TYPE S_ILValues_To_PC_Struct :
STRUCT
	PARAM000:REAL ;// 注入线法拉第筒温度节点01（℃） 
	PARAM001:REAL ;// 内靶温度节点02（℃） 
	PARAM002:REAL ;// 引出法拉第筒温度节点03（℃） 
	PARAM003:REAL ;// 温度节点04（℃） 
	PARAM004:REAL ;// 温度节点05（℃）
	PARAM005:REAL ;// 温度节点06（℃） 
	PARAM006:REAL ;// 温度节点07（℃） 
	PARAM007:REAL ;// 温度节点08（℃） 
	PARAM008:BOOL ;// 已经移去接地 
	PARAM009:BOOL ;// 地坑栅栏门已经关闭 
	PARAM010:BOOL ;// 加速器已合盖 
	PARAM011:BOOL ;// 无源节点01 
	PARAM012:BOOL ;// 无源节点02 
	PARAM013:BOOL ;// 离子源角阀2联锁开 
	PARAM014:BOOL ;// 离子源角阀2联锁关 
	PARAM015:BOOL ;// 注入线放气阀联锁开 
	PARAM016:BOOL ;// 注入线放气阀联锁关 
	PARAM017:BOOL ;// 离子源干泵联锁开 
	PARAM018:BOOL ;// 离子源干泵联锁关 
	PARAM019:BOOL ;// 离子源分子泵V1联锁开 
	PARAM020:BOOL ;// 离子源分子泵V1联锁关 
	PARAM021:BOOL ;// 离子源分子泵V3联锁开 
	PARAM022:BOOL ;// 离子源分子泵V3联锁关 
	PARAM023:BOOL ;// 离子源分子泵V4联锁开 
	PARAM024:BOOL ;// 离子源分子泵V4联锁关 
	PARAM025:BOOL ;// 冷泵隔断阀1联锁开 
	PARAM026:BOOL ;// 冷泵隔断阀1联锁关 
	PARAM027:BOOL ;// 冷泵隔断阀2联锁开 
	PARAM028:BOOL ;// 冷泵隔断阀2联锁关 
	PARAM029:BOOL ;// 主真空角阀1联锁开 
	PARAM030:BOOL ;// 主真空角阀1联锁关 
	PARAM031:BOOL ;// 主真空放气阀联锁开 
	PARAM032:BOOL ;// 主真空放气阀联锁关
	PARAM033:BOOL ;// 主真空干泵联锁开 
	PARAM034:BOOL ;// 主真空干泵联锁关 
	PARAM035:BOOL ;// 主真空分子泵V2联锁开 
	PARAM036:BOOL ;// 主真空分子泵V2联锁关 
	PARAM037:BOOL ;// 冷泵前级阀1联锁开 
	PARAM038:BOOL ;// 冷泵前级阀1联锁关 
	PARAM039:BOOL ;// 冷泵1联锁开 
	PARAM040:BOOL ;// 冷泵1联锁关 
	PARAM041:BOOL ;// 冷泵前级阀2联锁开 
	PARAM042:BOOL ;// 冷泵前级阀2联锁关 
	PARAM043:BOOL ;// 冷泵2联锁开 
	PARAM044:BOOL ;// 冷泵2联锁关 
	PARAM045:BOOL ;// 束流线1角阀联锁开 
	PARAM046:BOOL ;// 束流线1角阀联锁关 
	PARAM047:BOOL ;// 束流线1放气阀联锁开 
	PARAM048:BOOL ;// 束流线1放气阀联锁关 
	PARAM049:BOOL ;// 束流线1干泵联锁开 
	PARAM050:BOOL ;// 束流线1干泵联锁关 
	PARAM051:BOOL ;// 束流线1分子泵V5联锁开 
	PARAM052:BOOL ;// 束流线1分子泵V5联锁关 
	PARAM053:BOOL ;// 束流线2角阀联锁开 
	PARAM054:BOOL ;// 束流线2角阀联锁关 
	PARAM055:BOOL ;// 束流线2放气阀联锁开 
	PARAM056:BOOL ;// 束流线2放气阀联锁关 
	PARAM057:BOOL ;// 束流线2干泵联锁开 
	PARAM058:BOOL ;// 束流线2干泵联锁关 
	PARAM059:BOOL ;// 束流线2分子泵V6联锁开 
	PARAM060:BOOL ;// 束流线2分子泵V6联锁关
	PARAM061:BOOL ;// 束流线3角阀联锁开 
	PARAM062:BOOL ;// 束流线3角阀联锁关 
	PARAM063:BOOL ;// 束流线3放气阀联锁开 
	PARAM064:BOOL ;// 束流线3放气阀联锁关 
	PARAM065:BOOL ;// 束流线3干泵联锁开 
	PARAM066:BOOL ;// 束流线3干泵联锁关 
	PARAM067:BOOL ;// 束流线3分子泵V7联锁开 
	PARAM068:BOOL ;// 束流线3分子泵V7联锁关 
	PARAM069:BOOL ;// 注入线隔断阀联锁拉开 
	PARAM070:BOOL ;// 注入线隔断阀联锁插入 
	PARAM071:BOOL ;// 注入线法拉第筒联锁拉开 
	PARAM072:BOOL ;// 注入线法拉第筒联锁插入 
	PARAM073:BOOL ;// 内靶联锁拉开 
	PARAM074:BOOL ;// 内靶联锁插入 
	PARAM075:BOOL ;// 束流线1隔断阀联锁开 
	PARAM076:BOOL ;// 束流线1隔断阀联锁关 
	PARAM077:BOOL ;// 束流线2隔断阀联锁开 
	PARAM078:BOOL ;// 束流线2隔断阀联锁关 
	PARAM079:BOOL ;// 束流线3隔断阀联锁开 
	PARAM080:BOOL ;// 束流线3隔断阀联锁关 
	PARAM081:BOOL ;// 引出法拉第筒联锁拉开 
	PARAM082:BOOL ;// 引出法拉第筒联锁插入 
	PARAM083:BOOL ;// 离子源高压电源联锁开 
	PARAM084:BOOL ;// 离子源高压电源联锁关 
	PARAM085:BOOL ;// 正偏转版电源联锁开 
	PARAM086:BOOL ;// 正偏转版电源联锁关 
	PARAM087:BOOL ;// 负偏转版电源联锁开 
	PARAM088:BOOL ;// 正偏转版电源联锁关 
END_STRUCT
END_TYPE

(* stored: Version 1.1.0.1, ProductVersion 3.1.4024.16
   DUT S_ILValues_To_PC_Struct: Id {132d7c5a-3ba4-4b52-9b00-3105aa1b9bce} *)
